TYPE "LubrValve_Pers"
VERSION : 0.1
// Block: LubrValve_Pers
   STRUCT
      Par : LubrValve_Par;
      ValvePumpCounter : Int;
      LubrReqCounter : LReal;
   END_STRUCT;

END_TYPE
